FUNCTION_BLOCK FB_MotorsReset
VAR_INPUT
	bExecute : BOOL;
END_VAR
VAR_OUTPUT
	bResetDone : BOOL;
	bResetError: BOOL;
END_VAR
VAR_IN_OUT
	Axis : AXIS_REF;
END_VAR
VAR
	fbReset	: MC_Reset;
	bReset	: BOOL := TRUE;
END_VAR

//Axis Reset
IF bExecute THEN
	fbReset(Axis := Axis, Execute := bReset, Done => bResetDone, Error => bResetError);
END_IF
IF bResetDone THEN
	bReset := FALSE;
END_IF

END_FUNCTION_BLOCK

(* stored: Version 1.1.0.1, ProductVersion 3.1.4024.12
   POU FB_MotorsReset: Id {7a3e4215-b5be-40fe-b889-7d70a5148238}, SpecialFunc None *)
